// Empty function block that implements an empty interface only.
FUNCTION_BLOCK FB_EmptyWithEmptyImpl
IMPLEMENTS I_Empty
VAR
END_VAR

END_FUNCTION_BLOCK

(* stored: Version 1.1.0.1, ProductVersion 3.1.4024.15
   POU FB_EmptyWithEmptyImpl: Id {141e27aa-bd04-454e-86d1-c16f0586b236}, SpecialFunc None *)
